TYPE ST_MotorParam :
STRUCT
	Unit : STRING;
	Set : INT;
	P: UINT;
	I: UINT;
	D: UINT;
END_STRUCT
END_TYPE

(* stored: Version 1.1.0.1, ProductVersion 3.1.4022.18
   DUT ST_MotorParam: Id {f2c83422-cc8e-4e0e-99e3-6c0f8ae0865f} *)
